INTERFACE I_JsonDeserializerChangedEvent EXTENDS I_Event

PROPERTY PUBLIC Target : I_JsonDeserializer
GET
END_GET
END_PROPERTY

END_INTERFACE

(* stored: Version 1.1.0.1, ProductVersion 3.1.4024.12
   Itf I_JsonDeserializerChangedEvent: Id {dad098ca-719a-4568-8744-6322a5303569}
   Property Target: Id {52c45db3-5c7b-4027-8dc8-b5a450bc3550}
   Get Get: Id {ba968a51-bdc7-4946-9b02-504882d9f01f} *)
